FUNCTION_BLOCK CNV_CTRL (* Basic Function Block Type *)
  (* Standard: 61499-2 *)
  (* Version 0.3, 2009-09-15, JHC, Holobloc Inc, Changed transition priorities. *)
  (* Version 0.2, 2003-12-04, JHC, Rockwell Automation, Renamed for better indexing. *)
  (* Version 0.1, 2002-11-05, JHC, Rockwell Automation, Corrected missing ST element in Algorithm REQ. *)
  (* Version 0.0, 2000-05-30, JHC, Rockwell Automation *)
  PACKAGE fb.rt.Conveyer;
  IMPORT fb.datatype.*;
  IMPORT fb.rt.*;
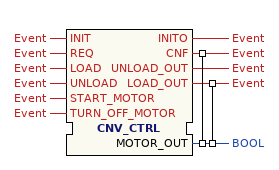
  EVENT_INPUT
    INIT; (* Initialization Request *)
    REQ; (* Normal Execution Request *)
    LOAD;
    UNLOAD;
    START_MOTOR;
    TURN_OFF_MOTOR;
  END_EVENT
  EVENT_OUTPUT
    INITO; (* Initialization Confirm *)
    CNF WITH MOTOR_OUT; (* Execution Confirmation *)
    UNLOAD_OUT;
    LOAD_OUT WITH MOTOR_OUT;
  END_EVENT
  VAR_OUTPUT
    MOTOR_OUT : BOOL;
  END_VAR
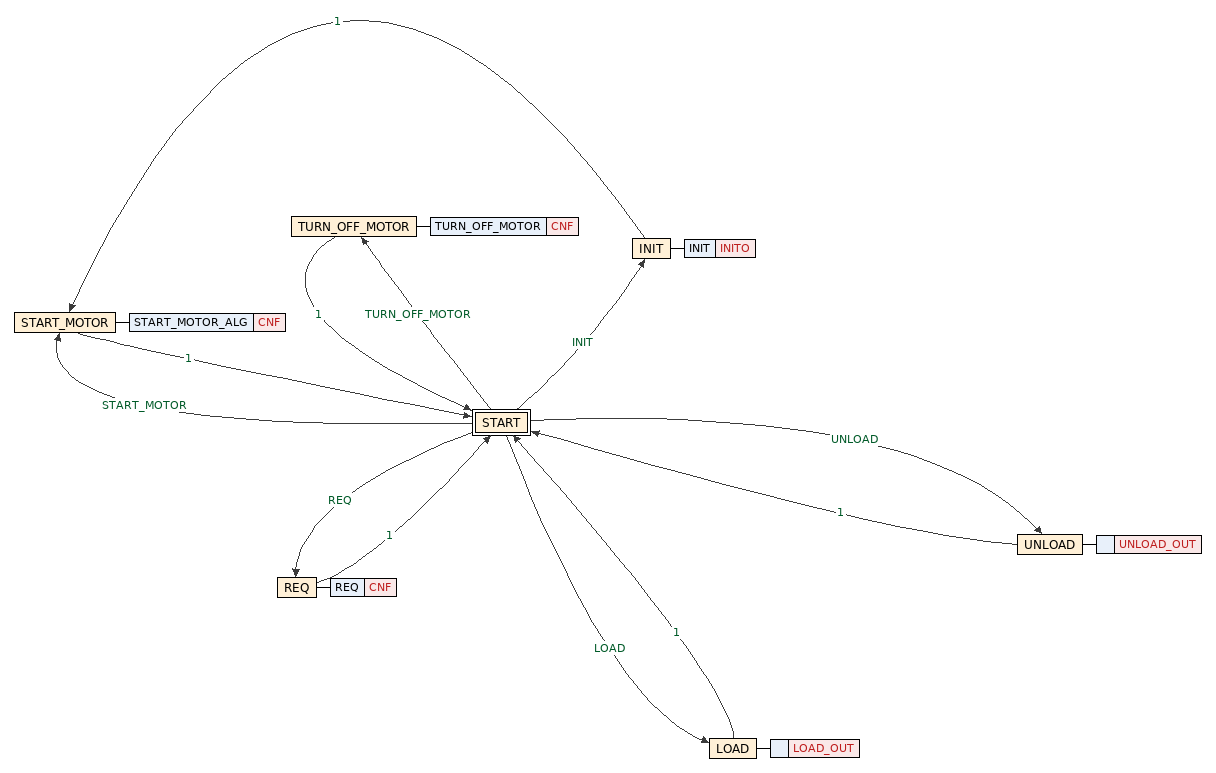
  EC_STATES
    START; (* Initial State *)
    INIT : INIT -> INITO; (* Initialization *)
    REQ : REQ -> CNF; (* Normal execution *)
    UNLOAD : -> UNLOAD_OUT;
    LOAD : -> LOAD_OUT;
    START_MOTOR : START_MOTOR_ALG -> CNF;
    TURN_OFF_MOTOR : TURN_OFF_MOTOR -> CNF;
  END_STATES
  EC_TRANSITIONS
    START TO REQ := REQ;
    START TO INIT := INIT;
    REQ TO START := 1;
    START TO UNLOAD := UNLOAD;
    UNLOAD TO START := 1;
    START TO LOAD := LOAD;
    LOAD TO START := 1;
    START TO START_MOTOR := START_MOTOR;
    START_MOTOR TO START := 1;
    TURN_OFF_MOTOR TO START := 1;
    START TO TURN_OFF_MOTOR := TURN_OFF_MOTOR;
    INIT TO START_MOTOR := 1;
  END_TRANSITIONS
  ALGORITHM INIT IN ST: (* Initialization algorithm *)
MOTOR_OUT := TRUE;
  END_ALGORITHM
  ALGORITHM REQ IN ST: (* Normally executed algorithm *)

  END_ALGORITHM
  ALGORITHM START_MOTOR_ALG IN ST:
MOTOR_OUT := TRUE;
  END_ALGORITHM
  ALGORITHM TURN_OFF_MOTOR IN ST:
MOTOR_OUT := FALSE;
  END_ALGORITHM
END_FUNCTION_BLOCK
